// TIA Portal V20 export
TYPE "typeSequenceControlNodeInterafceSTKJobInterfaceCommands"
// stored: Namespace Unit1.Em7
   STRUCT
      spare { ExternalWritable := 'False'} : Bool;
   END_STRUCT;
END_TYPE
